(* PLC project PacFramwork, Machine Expert Logic Builder V21.0.22.0, author roma_mirkevich *)
(* stored: creationDateTime 2024-02-07T15:48:44.9672837, version 0.0.0.0, modificationDateTime 2021-04-29T23:02:57.5377485 *)

TYPE PLC_STA : STRUCT
  CON2ERR : BOOL;  (* =1 - є помилка звязку з сусідні ПЛК в парі (для теплого резерування) *)
  PLC2STOP : BOOL;  (* =1 - спарений ПЛК в стопі (для теплого резерування) *)
  BLK : BOOL;  (* =1 – є хоча б один заблокований ВМ *)
  ALDIS : BOOL;  (* =1 – є хоча б одна відключена тривога *)
  DIOON : BOOL;  (* =1 - йде опитування по мережі (MODBUS або аналогічній) засобів віддаленого вводу/виводу *)
  DIOERR : BOOL;  (* =1 - є помилка на DIO *)
  b6 : BOOL;
  FRC : BOOL;  (* =1 – хоча б одна змінна форсована на будь якому рівні *)
  SMLALL : BOOL;  (* =1 – все в режимі в імітації, примушує усі CM перейти в режим імітації *)
  DISP : BOOL;  (* =1 – хоча б один елемент в режимі ручного управління *)
  FRC2 : BOOL;  (* =1 – є хоча б один форсований керівний елемент (рівня 2), клапан, двигун *)
  FRC1 : BOOL;  (* =1 – хоча б одна змінна форсована (рівня 1) *)
  SCN1 : BOOL;  (* =1 – перший скан *)
  FRC0 : BOOL;  (* =1 – хоча б одна змінна форсована (рівня 0) *)
  SML : BOOL;  (* =1 – хоча б один об’єкт в режимі імітації *)
  CMDACK : BOOL;  (* =1 - підтвердження команди, команда пройшла через весь цикл задачі і отримана усіма *)
END_STRUCT;
END_TYPE

TYPE PLC_ALM1 : STRUCT
  ALM : BOOL;  (* =1 - є активна тривога *)
  NWALM : BOOL;  (* =1 - є нова тривога *)
  ALMNACK : BOOL;  (* =1 - біт підтвердження тривоги *)
  WRN : BOOL;  (* =1 - є активне попередження *)
  NWWRN : BOOL;  (* =1 - є нове попередження *)
  WRNNACK : BOOL;  (* =1 - біт підтвердження попередження *)
  BAD : BOOL;  (* =1 - є активна тривога недостовірності даних *)
  NWBAD : BOOL;  (* =1 - є нова тривога недостовірності даних *)
  BADNACK : BOOL;  (* =1 - біт підтвердження тривоги недостовірності даних *)
  EMCYSTP : BOOL;  (* =1, аварійний зупин (грибок) *)
  STP2RUN : BOOL;  (* =1, момент переходу з аварійного зупину в роботу *)
  CON2ERR : BOOL;  (* =1 - є помилка звязку з сусідні ПЛК в парі (для теплого резерування) *)
  PLC2STOP : BOOL;  (* =1 - спарений ПЛК в стопі (для теплого резерування) *)
  DIOERR : BOOL;  (* =1 - є помилка DIO *)
  PLCERR : BOOL;  (* =1 – є апаратна помилка (ПЛК) *)
  CONHIERR : BOOL;  (* =1 – єпомилка звязку з верхнім рівнем *)
END_STRUCT;
END_TYPE

TYPE PLS : STRUCT
  P100MS : BOOL;  (* 100 мс *)
  P200MS : BOOL;  (* 200 мс *)
  P500MS : BOOL;  (* 500 мс *)
  P1S : BOOL;  (* 1 с *)
  P2S : BOOL;  (* 2 с *)
  P5S : BOOL;  (* 5 с *)
  P10S : BOOL;  (* 10 с *)
  P60S : BOOL;  (* 1 хв *)
  M1S : BOOL;  (* меандр з періодом 1 с (0.5 с + 0.5 с) *)
  M2S : BOOL;  (* меандр з періодом 2 с (1 с + 1 с) *)
  b10 : BOOL;
  b11 : BOOL;
  NEWMIN : BOOL;  (* =1 (на один цикл основної задачі) – початок хвилини *)
  NEWHR : BOOL;  (* =1 (на один цикл основної задачі) – початок години *)
  NEWDAY : BOOL;  (* =1 (на один цикл основної задачі) – початок доби *)
  NEWSHIFT : BOOL;  (* =1 (на один цикл основної задачі) – початок зміни *)
END_STRUCT;
END_TYPE

TYPE PLC_CFG : STRUCT
  ID : UINT;  (* Унікальний ідентифікатор *)
  CLSID : UINT;  (* 1621xx *)
  STA : PLC_STA;  (* набір біт типу PLC_STA *)
  CMD : UINT;  (* Команди з HMI *)
  CMDPRG : UINT;  (* Команди з програмного керування (побітові) *)
  PRM1 : UINT;  (* дискретні параметри *)
  PRM2 : UINT;  (* дискретні параметри *)
  PLS : PLS;  (* бітові міандри *)
  ALM1 : PLC_ALM1;  (* біти алармів *)
  ALM2 : INT;  (* біти алармів *)
  STEP1 : INT;  (* крок основної програми *)
  T_STEP1 : INT;  (* час кроку основної програми обробки, в (с) *)
  MSG : UDINT;  (* для формування повідомлень, може бути як бітовим (32 повідомлення), так і числовим (за номером); передбачається, що повідомлення буде скидуватися в 0 автоматично через певний час (не менш ніж 2 інтервали опитування з HMI) *)
  TQ : UDINT;  (* загальний час з початку 1-го циклу контролера (в секундах) *)
  TQM : UDINT;  (* загальний час роботи ПЛК з моменту пуску (в хвилинах) *)
  DICNT : INT;  (* кількість наявних каналів DI *)
  DOCNT : INT;  (* кількість наявних каналів DO *)
  AICNT : INT;  (* кількість наявних каналів AI *)
  AOCNT : INT;  (* кількість наявних каналів AO *)
  NOW : ARRAY[0..3] OF INT;  (* плинний час астрономічний час в BCD форматі: NOW[0] seconds,-- (16ss,--) NOW[1] hour, minute (16hhmm) NOW[2] month, day (16mmdd) NOW[3] year (16yyyy) *)
  SHIFTPARA : ARRAY[0..3] OF INT;  (* Години передачі змін (максимум 3 зміни): SHIFT[0] – кількість змін SHIFT[1] – передача 1-ї зміни (BCD 16hhmm) SHIFT[2] – передача 2-ї зміни (BCD 16hhmm) SHIFT[3] – передача 3-ї зміни (BCD 16hhmm) *)
  SHIFTNMB : UINT;  (* номер активної зміни *)
  CNTALM : UINT;  (* лічильник кількості активних тривог аварія *)
  CNTWRN : UINT;  (* лічильник кількостіактивних тривог попередження *)
  CNTBAD : UINT;  (* лічильник кількостіактивних тривог недостовірність *)
  CNTFRC : UINT;  (* лічильник кількостіфорсованих об'єктів *)
  CNTMAN : UINT;  (* лічильник кількості ВМ в ручному режимі *)
  TSK_LTIME : UINT;  (* плинний (останній) час задачі в мілісекундах *)
  TSK_MAXTIME : UINT;  (* максимальний час задачі в мілісекундах *)
  STA_PERM : UINT;  (* повторює STA, який був на початку виклику функції *)
  ALM1_PERM : UINT;  (* повторює ALM1, який був на початку виклику функції *)
  CNTALM_PERM : UINT := 0;  (* лічильник кількості активних тривог аварія *)
  CNTWRN_PERM : UINT := 0;  (* лічильник кількостіактивних тривог попередження *)
  CNTBAD_PERM : UINT := 0;  (* лічильник кількостіактивних тривог недостовірність *)
  CNTFRC_PERM : UINT := 0;  (* лічильник кількостіфорсованих об'єктів *)
  CNTMAN_PERM : UINT := 0;  (* лічильник кількості ВМ в ручному режимі *)
  MODULSCNT : INT;  (* кількість модулів *)
  NOWns : UDINT;  (* нс (наносекунди) для плинного астрономічного часу *)
  TQMS : UDINT;  (* мілісекундний лічильник, скидається при старті або після переповнення *)
END_STRUCT;
END_TYPE

FUNCTION_BLOCK PLCFN
  VAR_IN_OUT
    PLC : PLC_CFG;
  END_VAR
  VAR_GLOBAL
    TMBITS_PREV : INT;  (* попереднє значення таймерних меандрів *)
    MEM_RT : LREAL;  (* память для вимірювання часу циклу *)
    FirstScan : BOOL;
    NextScan : BOOL;
    Clock_10Hz : BOOL;
    Clock_5Hz : BOOL;
    Clock_2Hz : BOOL;
    Clock_1Hz : BOOL;
    Clock_0_5Hz : BOOL;
    BLINK_10Hz : BLINK;
    BLINK_5Hz : BLINK;
    BLINK_2Hz : BLINK;
    BLINK_1Hz : BLINK;
    BLINK_0_5Hz : BLINK;
    iecResult : RTS_IEC_RESULT;
    pIecInfo : POINTER TO CmpIecTask.Task_Info2;
    LocalTime_ofset : INT := 2;
  END_VAR
  VAR_TEMP
    TMBITS_CUR : INT;
    i : INT;
    NOW : SYSTIMEDATE;
  END_VAR

            	IF PLC.STA.CMDACK THEN
	    PLC.CMD := 0;
	END_IF;
	PLC.STA.CMDACK := (PLC.CMD <> 0 AND NOT PLC.STA.CMDACK);
	
	(*--------------------------------- Визначення біту першого скану*)
	
	IF NOT FirstScan AND NOT NextScan THEN
		FirstScan := TRUE;
		NextScan:=TRUE;
	ELSE
		FirstScan := FALSE;
	END_IF


	
	PLC.STA.SCN1 := FirstScan;
	IF PLC.STA.SCN1 THEN (*при першому скані*)
	    PLC.ID := 1;             (*Ідентифікатор завжди 1*)
	    PLC.CLSID := 16#2100;    (*Клас завжди 162100*)
	    PLC.TQ := 0;
	    TMBITS_CUR := 0;
	    TMBITS_PREV := 0;
		PLC.TQMS := 0;
	END_IF;
	
	PLC.STA_PERM.0 := PLC.STA.CON2ERR;
	PLC.STA_PERM.1 := PLC.STA.PLC2STOP;
	PLC.STA_PERM.2 := PLC.STA.BLK;
	PLC.STA_PERM.3 := PLC.STA.ALDIS;
	PLC.STA_PERM.4 := PLC.STA.DIOON;
	PLC.STA_PERM.5 := PLC.STA.DIOERR;
	PLC.STA_PERM.6 := PLC.STA.b6;
	PLC.STA_PERM.7 := PLC.STA.FRC;
	PLC.STA_PERM.8 := PLC.STA.SMLALL;
	PLC.STA_PERM.9 := PLC.STA.DISP;
	PLC.STA_PERM.10 := PLC.STA.FRC2;
	PLC.STA_PERM.11 := PLC.STA.FRC1;
	PLC.STA_PERM.12 := PLC.STA.SCN1;
	PLC.STA_PERM.13 := PLC.STA.FRC0;
	PLC.STA_PERM.14 := PLC.STA.SML;
	PLC.STA_PERM.15 := PLC.STA.CMDACK;
	
	PLC.ALM1_PERM.0 := PLC.ALM1.ALM;
	PLC.ALM1_PERM.1 := PLC.ALM1.NWALM;
	PLC.ALM1_PERM.2 := PLC.ALM1.ALMNACK;
	PLC.ALM1_PERM.3 := PLC.ALM1.WRN;
	PLC.ALM1_PERM.4 := PLC.ALM1.NWWRN;
	PLC.ALM1_PERM.5 := PLC.ALM1.WRNNACK;
	PLC.ALM1_PERM.6 := PLC.ALM1.BAD;
	PLC.ALM1_PERM.7 := PLC.ALM1.NWBAD;
	PLC.ALM1_PERM.8 := PLC.ALM1.BADNACK;
	PLC.ALM1_PERM.9 := PLC.ALM1.EMCYSTP;
	PLC.ALM1_PERM.10 := PLC.ALM1.STP2RUN;
	PLC.ALM1_PERM.11 := PLC.ALM1.CON2ERR;
	PLC.ALM1_PERM.12 := PLC.ALM1.PLC2STOP;
	PLC.ALM1_PERM.13 := PLC.ALM1.DIOERR;
	PLC.ALM1_PERM.14 := PLC.ALM1.PLCERR;
	PLC.ALM1_PERM.15 := PLC.ALM1.CONHIERR;
	
	
	(*--------------------------------- таймерні біти та лічильники*)
	BLINK_10Hz(enable:=TRUE, timelow:=T#50MS, timehigh:=T#50MS, out=>Clock_10Hz);
	BLINK_5Hz(enable:=TRUE, timelow:=T#100MS, timehigh:=T#100MS, out=>Clock_5Hz);
	BLINK_2Hz(enable:=TRUE, timelow:=T#250MS, timehigh:=T#250MS, out=>Clock_2Hz);
	BLINK_1Hz(enable:=TRUE, timelow:=T#500MS, timehigh:=T#500MS, out=>Clock_1Hz);
	BLINK_0_5Hz(enable:=TRUE, timelow:=T#1000MS, timehigh:=T#1000MS, out=>Clock_0_5Hz);
	
	(*плинні значення*)
	TMBITS_CUR.0 := Clock_10Hz;         // 100MS 
	TMBITS_CUR.1 := Clock_5Hz;        // 200MS
	TMBITS_CUR.2 := Clock_2Hz;        // 500MS
	TMBITS_CUR.3 := Clock_1Hz;      // 1S
	TMBITS_CUR.7 := PLC.NOW[0] > 16#29; //min
	
	(*відловлювання імпульсів необхідних часових періодів*)
	PLC.PLS.P100MS := TMBITS_CUR.0 AND NOT TMBITS_PREV.0; (*100 мс *)
	PLC.PLS.P200MS := TMBITS_CUR.1 AND NOT TMBITS_PREV.1; (*200 мс*)
	PLC.PLS.P500MS := TMBITS_CUR.2 AND NOT TMBITS_PREV.2; (*500 мс*)
	PLC.PLS.P1S := TMBITS_CUR.3 AND NOT TMBITS_PREV.3; (*1 с*)
	PLC.PLS.P60S := TMBITS_CUR.7 AND NOT TMBITS_PREV.7; (*1 хв*)
	(*підрахунок кількості секунд і хвилин*)
	IF PLC.PLS.P1S THEN
	    PLC.TQ := PLC.TQ + 1;
	END_IF;  (*загальний час з початку 1-го циклу контролера (в секундах)*)
	IF PLC.TQ > 16#7FFF_FFFF THEN
	    PLC.TQ := 16#7FFF_FFFF;
	END_IF;
	IF PLC.PLS.P60S AND NOT PLC.STA.SCN1 THEN
	    PLC.TQM := PLC.TQM + 1;
	END_IF; (*загальний час роботи ПЛК з моменту пуску (в хвилинах)*)
	IF PLC.TQM > 16#7FFF_FFFF THEN
	    PLC.TQM := 16#7FFF_FFFF;
	END_IF;
	
	(*розрахунок інших часових періодів*)
	PLC.PLS.P2S := (PLC.TQ MOD 2) = 0 AND PLC.PLS.P1S;(*2 с*)
	PLC.PLS.P5S := (PLC.TQ MOD 5) = 0 AND PLC.PLS.P1S;(*5 с*)
	PLC.PLS.P10S := (PLC.TQ MOD 10) = 0 AND PLC.PLS.P1S;(*10 с*)
	
	(* меандри *)
	PLC.PLS.M1S := Clock_1Hz;  (*меандр з періодом 1 с (0.5 с + 0.5 с)*)
	PLC.PLS.M2S := Clock_0_5Hz;(*меандр з періодом 2 с (1 с + 1 с) *)
	
	(* астрономічний час *)
	SysTimeRtcConvertUtcToDate(dwTimestampUtc:= GetRTC()+LocalTime_ofset*3600, pDate:=NOW );
	PLC.NOW[0] := INT_TO_BCD(NOW.wSECOND); //NOW[0] seconds,-- (16ss,--)
	PLC.NOW[1] := SHL(INT_TO_BCD(NOW.wHOUR), 8) OR INT_TO_BCD(NOW.wMINUTE);//16hhmm
	PLC.NOW[2] := SHL(INT_TO_BCD(NOW.wMONTH), 8) OR INT_TO_BCD(NOW.wDAY);  //16mmdd
	PLC.NOW[3] := SHL(INT_TO_BCD(NOW.wYEAR / 100), 8) OR INT_TO_BCD(NOW.wYEAR MOD 100);; //16yyyy
	PLC.NOWns := INT_TO_BCD(now.wMilliseconds)*1000000;
	(* початок години *)
	PLC.PLS.NEWHR := (PLC.NOW[1] AND 16#00FF) = 0 (*хвилини*)AND PLC.PLS.P60S (*один раз за хвилину*);
	
	(* початок доби*)
	PLC.PLS.NEWDAY := PLC.NOW[1] = 0 (*години_хвилини*)AND PLC.PLS.P60S (*один раз за хвилину*);
	
	(*початок зміни*)
	IF PLC.SHIFTPARA[0] < 1 OR PLC.SHIFTPARA[0] > 3 THEN
	    PLC.SHIFTPARA[0] := 2;
	END_IF;(*коректність кількості змін*)
	PLC.PLS.NEWSHIFT := FALSE; (*скидуємо біт початку зміни*)
	FOR i := 1 TO PLC.SHIFTPARA[0] DO
	    (*хоча б одна з устоавок змін спрацювала*)
	    PLC.PLS.NEWSHIFT := PLC.PLS.NEWSHIFT OR (PLC.SHIFTPARA[i] = PLC.NOW[1] (*години хвилин*)AND PLC.PLS.P60S (*один раз за хвилину*));
	END_FOR;
	
	TMBITS_PREV := TMBITS_CUR;(*збереження попередніх значень*)
	
	(*----------- визначеня зміни*)
	IF PLC.SHIFTPARA[0] > 3 OR PLC.SHIFTPARA[0] < 2 THEN
	    PLC.SHIFTPARA[0] := 3;
	END_IF;(*якщо кількість змін >3 або <1 - робимо 3*)
	IF PLC.NOW[1] >= PLC.SHIFTPARA[1] AND (PLC.NOW[1] < PLC.SHIFTPARA[2] OR PLC.SHIFTPARA[2] = 16#0000) THEN (*1-ша зміна*)
	    PLC.SHIFTNMB := 1;
	ELSE (*2-га або 3-тя*)
	    IF PLC.SHIFTPARA[0] = 2 THEN (*якщо в 2 зміни*)
	        PLC.SHIFTNMB := 2;
	    ELSE (*якщо 3 зміни*)
	        IF PLC.NOW[1] >= PLC.SHIFTPARA[2] AND (PLC.NOW[1] < PLC.SHIFTPARA[3] OR PLC.SHIFTPARA[3] = 16#0000) THEN
	            PLC.SHIFTNMB := 2;
	        ELSE
	            PLC.SHIFTNMB := 3;
	        END_IF;
	    END_IF;
	END_IF;
	(*----------- *)
	
	(*цикли*)
	pIecInfo := IecTaskGetInfo3(hIecTask := IecTaskGetCurrent(pResult := ADR(iecResult)), pResult := ADR(iecResult));
	PLC.TSK_LTIME := DWORD_TO_UINT(pIecInfo^.dwCycleTime / 1000);
	
	
	IF NOT FirstScan THEN
	    //обмеження 
	    IF PLC.TSK_MAXTIME > 3000 THEN
	        PLC.TSK_MAXTIME := 0;
	    END_IF;
	    IF PLC.TSK_MAXTIME < PLC.TSK_LTIME THEN
	        PLC.TSK_MAXTIME := PLC.TSK_LTIME;
	    END_IF;
	ELSE
	    PLC.TSK_MAXTIME := 0;
	END_IF;
	PLC.TQMS := PLC.TQMS + PLC.TSK_LTIME;//лічильник в мс
	
	(*скидання статусів і тривог*)
	PLC.STA.BLK := false;
	PLC.STA.ALDIS := false;
	PLC.STA.FRC := false;
	PLC.STA.SMLALL := false;
	PLC.STA.DISP := false;
	PLC.STA.FRC2 := false;
	PLC.STA.FRC1 := false;
	PLC.STA.FRC0 := false;
	PLC.STA.SML := false;
	
	PLC.ALM1.ALM := 0;
	PLC.ALM1.NWALM := 0;
	PLC.ALM1.ALMNACK := 0;
	PLC.ALM1.WRN := 0;
	PLC.ALM1.NWWRN := 0;
	PLC.ALM1.WRNNACK := 0;
	PLC.ALM1.BAD := 0;
	PLC.ALM1.NWBAD := 0;
	PLC.ALM1.BADNACK := 0;
	PLC.ALM1.EMCYSTP := 0;
	PLC.ALM1.STP2RUN := 0;
	PLC.ALM1.CON2ERR := 0;
	PLC.ALM1.PLC2STOP := 0;
	PLC.ALM1.DIOERR := 0;
	PLC.ALM1.PLCERR := 0;
	PLC.ALM1.CONHIERR := 0;
	
	(*запамятовування лічильників*)
	PLC.CNTALM_PERM := PLC.CNTALM;
	PLC.CNTWRN_PERM := PLC.CNTWRN;
	PLC.CNTBAD_PERM := PLC.CNTBAD;
	PLC.CNTFRC_PERM := PLC.CNTFRC;
	PLC.CNTMAN_PERM := PLC.CNTMAN;
	
	(*скидання лічильників*)
	PLC.CNTALM := 0;
	PLC.CNTWRN := 0;
	PLC.CNTBAD := 0;
	PLC.CNTFRC := 0;
	PLC.CNTMAN := 0;
          
END_FUNCTION_BLOCK
